FUNCTION_BLOCK STARTandSTOP (* Basic Function Block Type *)
  (* Standard: 61499-2 *)
  (* Version 0.0, 05/07/2022, Etienne, Schneider Electric, Template *)
  PACKAGE Main;
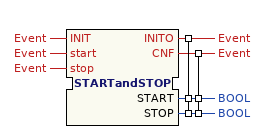
  EVENT_INPUT
    INIT; (* Initialization Request *)
    start;
    stop;
  END_EVENT
  EVENT_OUTPUT
    INITO WITH START, STOP; (* Initialization Confirm *)
    CNF WITH START, STOP; (* Execution Confirmation *)
  END_EVENT
  VAR_OUTPUT
    START : BOOL; (* Output event qualifier *)
    STOP : BOOL;
  END_VAR
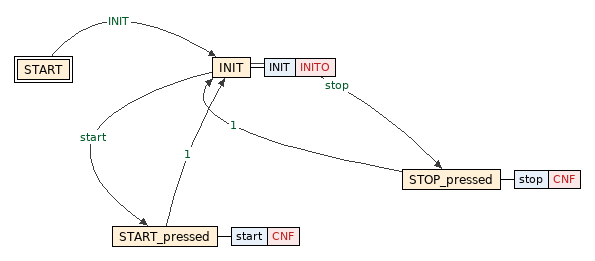
  EC_STATES
    START; (* Initial State *)
    INIT : INIT -> INITO; (* Initialization *)
    START_pressed : start -> CNF;
    STOP_pressed : stop -> CNF;
  END_STATES
  EC_TRANSITIONS
    START TO INIT := INIT;
    START_pressed TO INIT := 1;
    STOP_pressed TO INIT := 1;
    INIT TO START_pressed := start;
    INIT TO STOP_pressed := stop;
  END_TRANSITIONS
  ALGORITHM INIT IN ST: (* Initialization algorithm *)
;
START:=FALSE;
STOP:=FALSE;
  END_ALGORITHM
  ALGORITHM start IN ST:
;
START:=TRUE;
  END_ALGORITHM
  ALGORITHM stop IN ST:
;
STOP:=TRUE;
  END_ALGORITHM
END_FUNCTION_BLOCK
